{attribute 'qualified_only'}
{attribute 'strict'}
{attribute 'to_string'}
TYPE E_LogDebugLevel :
(
	invlid := 0,
	testing,
	commissioning,
	production
) UDINT;
END_TYPE

(* stored: Version 1.1.0.1
   DUT E_LogDebugLevel: Id {eab72703-e8d4-4809-b2c9-afc6803e5621} *)
